// TIA Portal V20 export
DATA_BLOCK "DB_OPC_State"   // DB112
// stored: InstanceOfName FB_OPC_State, InstanceOfType FB
"FB_OPC_State"
   // VAR
   //    sAutoReq : Bool;
   //    sSemiAutoReq : Bool;
   //    sManuReq : Bool;
   //    sRT_AutoReq : R_TRIG;
   //    sRT_SemiAutoReq : R_TRIG;
   //    sRT_ManuReq : R_TRIG;
   // END_VAR
BEGIN
END_DATA_BLOCK
